PROGRAM Version
VAR
END_VAR

(*
1.0.1.1:	Boido	010120

Added VersionLib and Verstion.txt to the project.

1.0.2.2:	Boido	020120

Version.txt replaced with Version PRG

*)

END_PROGRAM

(* stored: Version 1.1.0.1, ProductVersion 3.1.4024.0
   POU Version: Id {daa0953d-9a0f-43c6-80ef-58b14101c0d8}, SpecialFunc None *)
